FUNCTION_BLOCK StopMotorsTask EXTENDS TcoCore.TcoTask 
VAR
    {attribute 'hide'} 
	_progress : INT := 0;
    {attribute 'hide'} 
	_infoTimer :  TON;
    {attribute 'hide'} 
	_errorTimer :  TON;
    {attribute 'hide'} 
	_varInfo : __SYSTEM.VAR_INFO;
    {attribute 'hide'} 
	_sb : TcoCore.StringBuilder;
END_VAR

VAR_IN_OUT
    inoConfig 	: TcoIrc5_Config_v_1_x_x;
	inoControl 	: TcoIrc5_Control_v_1_x_x;
	inoStatus 	: TcoIrc5_Status_v_1_x_x;	
END_VAR

IF Execute() THEN 
	IF _progress = 0 THEN
		IF NOT __ISVALIDREF(inoControl) THEN
			_varInfo :=__VARINFO(inoControl);
			Messenger.Programming(_sb.Clear().Append('<#Invalid reference: #>').Append(_varInfo.Symbol).ToString()).Pin();
		ELSIF NOT __ISVALIDREF(inoConfig) THEN                                                  
			_varInfo :=__VARINFO(inoConfig);                                                    
			Messenger.Programming(_sb.Clear().Append('<#Invalid reference: #>').Append(_varInfo.Symbol).ToString()).Pin();
		ELSIF NOT __ISVALIDREF(inoStatus) THEN                                                  
			_varInfo :=__VARINFO(inoStatus);                                                    
			Messenger.Programming(_sb.Clear().Append('<#Invalid reference: #>').Append(_varInfo.Symbol).ToString()).Pin();
		ELSE
			_progress := _progress + 1;
		END_IF

	END_IF
	IF _progress = 1 THEN
	
		
		inoControl.MotorOff := TRUE ;
		
		IF inoStatus.State.MotorOffState AND NOT inoStatus.State.SystemInputBusy THEN
			inoControl.MotorOff :=FALSE;
			_progress:=0;
		END_IF
	END_IF
    DoneWhen(inoStatus.State.MotorOffState AND NOT inoStatus.State.SystemInputBusy);
    CallTimers(TRUE);
	
	THIS^.ThrowWhen(_errorTimer.Q);
	
END_IF;

METHOD CallTimers
VAR_INPUT
	inValue : BOOL;
END_VAR
IF  __ISVALIDREF(inoConfig) THEN  
_infoTimer(IN := inValue, PT := THIS^.inoConfig.InfoTime);
_errorTimer(IN := inValue, PT := THIS^.inoConfig.ErrorTime);
END_IF;
END_METHOD

METHOD PUBLIC FB_init : BOOL
VAR_INPUT
    bInitRetains : BOOL; // if TRUE, the retain variables are initialized (warm start / cold start)
    bInCopyCode : BOOL; // if TRUE, the instance afterwards gets moved into the copy code (online change)
  	ParentObject : ITcoObject;	
END_VAR
END_METHOD

(*~
	<docu>
		<summary>
			Executes when task is aborted.
		</summary>			
	</docu>	
~*)
METHOD PROTECTED OnAbort
IF  __ISVALIDREF(inoStatus) THEN   THIS^.inoStatus.ActionDescription := '<#Start at Main was aborted, while not yet completed!#>';END_IF; 
inoControl.MotorOff :=FALSE;
END_METHOD

(*~
	<docu>
		<summary>
			Executes when task reaches the ```Done``` state .
		</summary>			
	</docu>	
~*)
METHOD PROTECTED OnDone
IF  __ISVALIDREF(inoStatus) THEN  THIS^.inoStatus.ActionDescription := '<#Stop motors was completed successfully.#>';END_IF;
END_METHOD

(*~
	<docu>
		<summary>
			Executes when task reaches the ```Error``` state.
			<para>
				Do not confuse with <see cref="PlcDocu.TcoCore.TcoTask.WhileError()"/>, that is called cyclically until '''Error''' state is left.
			</para>
		</summary>			
	</docu>	
~*)
METHOD PROTECTED OnError
IF  __ISVALIDREF(inoStatus) THEN   THIS^.inoStatus.ActionDescription := '<#Stop motors finished with error.#>'; END_IF;
END_METHOD

METHOD PROTECTED OnStart
IF  __ISVALIDREF(inoStatus) THEN  THIS^.inoStatus.ActionDescription := '<#Stop motors started.#>'; END_IF;
END_METHOD

(*~
	<docu>
		<summary>
			Restores this instance to the Ready state. Can be called explicitly or from within one of the restore mechanisms.
			<para>
				See also <see cref="PlcDocu.TcoCore.TcoTask.AutoRestorable()"/>
			</para>
		</summary>			
	</docu>	
~*)
METHOD Restore : ITcoRestorable
SUPER^.Restore();
_progress := 0;
CallTimers(FALSE);
Messenger.UnPin();
inoControl.MotorOff :=FALSE;
END_METHOD

END_FUNCTION_BLOCK

(* stored: Version 1.1.0.1, ProductVersion 3.1.4024.12
   POU StopMotorsTask: Id {cacb6202-7142-04df-0a56-64e9983344e3}, SpecialFunc None
   Method CallTimers: Id {bf5361e4-1b30-020c-2163-a798e7e162d6}
   Method FB_init: Id {c4635951-a02c-07b8-14cb-6118e1da4fe7}
   Method OnAbort: Id {21fe370e-1acf-0049-2670-d27ac9c32c0f}
   Method OnDone: Id {77832d71-89c0-0f34-3e9c-a083b2686171}
   Method OnError: Id {44292be8-8f48-026a-02c2-425eed01693e}
   Method OnStart: Id {64c6ed6e-e5f5-03c6-11ee-d2694369b6d8}
   Method Restore: Id {88ec3d47-bb9a-0940-346e-0e635e4eec04} *)
